// This function has been automatically generated from the project information.
{attribute 'signature_flag' := '1073741824'}
{attribute 'TcGenerated'}
{attribute 'no-analysis'}
FUNCTION F_GetCompany : WSTRING
VAR_INPUT
	
END_VAR

F_GetCompany := "ekvip automation GmbH";

END_FUNCTION

(* stored: Version 1.1.0.1
   POU F_GetCompany: Id {4a339fc2-b624-4dcc-9341-7070b7927981}, SpecialFunc None *)
